TYPE AX5000_S_0007 :
STRUCT
	Feedvack_acquisition_capture_point:UINT;
END_STRUCT
END_TYPE

(* stored: Version 1.1.0.1, ProductVersion 3.1.4024.3
   DUT AX5000_S_0007: Id {64e982b7-daec-4bed-a800-737463879306} *)
